TYPE ST_EL6070 :
STRUCT
	
	// TERMINAL - EL6070	EtherCAT Terminal, license key FOR TwinCAT 3.1  (Term 2)
	sTerminalName                                           :   STRING(200):= 'EtherCAT Terminal, license key FOR TwinCAT 3.1';
	stTerminalInfo											: 	ST_Terminal_Info;

END_STRUCT
END_TYPE

(* stored: Version 1.1.0.1, ProductVersion 3.1.4024.13
   DUT ST_EL6070: Id {1689a7e5-5088-4759-b76a-5c06002d039f} *)
